// TwinCAT 3 PLC project Aufgabe5
// ProgramVersion: 3.1.4023.0
// libraries:
//   Tc2_Standard, * (Beckhoff Automation GmbH)
//   Tc2_System, * (Beckhoff Automation GmbH)
//   Tc3_Module, * (Beckhoff Automation GmbH)
// project tree:
//   / PlcTask.TcTTO
//   POUs/ Fb_EdgeDetector.TcPOU, FB_Integrator.TcPOU, FB_LowpassFilter.TcPOU, Fb_MeanCalculatorWForgettingFactor.TcPOU, FB_PWM.TcPOU (not stored), FB_SecondOrderHold.TcPOU, F_Sine.TcPOU, F_Square.TcPOU, MAIN.TcPOU
// real-time tasks:
//   TASK PlcTask: cycle T#10ms, priority 20, ADS port 350

CONFIGURATION Aufgabe5
    RESOURCE PLC ON TwinCAT3
        TASK PlcTask(INTERVAL := T#10ms, PRIORITY := 20);
        PROGRAM MAIN WITH PlcTask : MAIN;
    END_RESOURCE
END_CONFIGURATION

// ---- POUs/MAIN.TcPOU
PROGRAM MAIN
VAR
	// sinus
	u_k_sin			: REAL;				// u_k sinus
	u_k_sin_f		: REAL;				// u_k sinus filtered
	w_sin			: REAL := (1/tau);	// Frequenz
	lowPassSin		: FB_LowpassFilter;
	// constant
	u_k_cst			: REAL;				// u_k constant
	u_k_cst_f		: REAL;				// u_k constant filtered
	lowPassConst	: FB_LowpassFilter;
	// pt2
	d				: REAL		:= 0.2;
	w0				: REAL		:= 10;
	u_k_pt2_f		: REAL;				// u_k pt2 filtered
	secondOrder		: FB_SecondOrderHold;
	// integrator
	pwm				: FB_PWM;
	integrator		: FB_Integrator;
	dutyCyclePct	: REAL		:= 25; 	// duty cycle for PWM in %
	pwmOut			: REAL;				// pwm signal
	integratorOut	: REAL;				// integrated PWM signal
	
	actTime			: REAL 	:= 0;		// time increment
	
END_VAR
VAR CONSTANT
	sampleTime		: REAL	:= 0.001;	// Abtastzeit	
	tau 			: REAL	:= 0.1;		// filter constant
END_VAR

// Integrator PWM
pwm(dutyPct := dutyCyclePct, ymin := 0, ymax := 5, w := 3.14, t := actTime);
pwmOut := pwm.y;
integrator(u_k := pwmOut, T := sampleTime);
integratorOut := integrator.y_k;

// Lowpass Sinus
u_k_sin := F_Sine(A := 1.0, yoff := 0.0, w := w_sin, t := actTime);
lowPassSin(u_k := u_k_sin, T := sampleTime, tau := tau);
u_k_sin_f := lowPassSin.y_k;

// PT2 with sinus
secondOrder(u_k := u_k_sin, T := sampleTime, d := d, w0 := w0);
u_k_pt2_f := secondOrder.y_k;

actTime := actTime + sampleTime;

END_PROGRAM

// ---- POUs/FB_LowpassFilter.TcPOU
FUNCTION_BLOCK FB_LowpassFilter
VAR_INPUT
	u_k		: REAL;
	T		: REAL;
	tau		: REAL;
END_VAR
VAR_OUTPUT
	y_k		: REAL;
END_VAR
VAR
	y_k_1	: REAL;
END_VAR

// limit tau
IF tau < 0.0001 THEN
	tau := 0.0001;
END_IF

y_k := tau / (T+tau) * y_k_1 + T / (T+tau) * u_k;
y_k_1 := y_k;

END_FUNCTION_BLOCK

// ---- POUs/FB_SecondOrderHold.TcPOU
FUNCTION_BLOCK FB_SecondOrderHold
VAR_INPUT
	u_k		: REAL; // Eingangswert
	T		: REAL;	// Zeitkonstante
	d		: REAL; // Daempfung
	w0		: REAL; // Eigenfrequenz 
END_VAR
VAR_OUTPUT
	y_k		: REAL; // Ausgangswert
END_VAR
VAR
	a		: REAL; // Variable fuer w0^2 * T^2
	b 		: REAL; // Variable fuer 2 * d * w0 * T
	y_k_1	: REAL; // letzer Ausgangswert
	y_k_2	: REAL; // vorletzer Ausgangswert
END_VAR

a := (w0 * w0) * (T * T);
b := 2 * d * w0 * T; 

y_k := (u_k*a + 2*y_k_1 + b*y_k_1 - y_k_2) / (1 + b + a); 

y_k_2 := y_k_1;
y_k_1 := y_k;

END_FUNCTION_BLOCK

// ---- POUs/FB_Integrator.TcPOU
FUNCTION_BLOCK FB_Integrator
VAR_INPUT
	u_k		: REAL;
	T		: REAL;
END_VAR
VAR_OUTPUT
	y_k		: REAL;
END_VAR
VAR
	y_k_1	: REAL;
END_VAR

y_k := u_k * T + y_k_1;
y_k_1 := y_k;

END_FUNCTION_BLOCK

// ---- POUs/F_Sine.TcPOU
FUNCTION F_Sine : REAL
VAR_INPUT
	A		: REAL;	// Amplitude
	yoff	: REAL; // offset
	w		: REAL; // Kreisfrequenz (rad/s)
	t		: REAL; // Time (s)
END_VAR
VAR
END_VAR

F_Sine := (A * SIN(w*t)) + yoff;

END_FUNCTION

// ---- POUs/Fb_EdgeDetector.TcPOU
FUNCTION_BLOCK INTERNAL Fb_EdgeDetector
VAR_INPUT
	inputValue		: BOOL;
END_VAR
VAR_OUTPUT
	risingEdge		: BOOL;
	fallingEdge		: BOOL;
	doublePress		: BOOL;
	triplePress		: BOOL;
END_VAR
VAR
	i_risingEdgCnt			: INT := 0;  		// internal var
	lastValue 				: BOOL;				// last value registered
	tlastPush				: TIME := TIME();	// time when last push happened
	tLastRising				: TIME := TIME();	// time when last rising edge happened
	tDebounce	    		: TIME := T#20MS;   // time to debounce input value
	tMultiPressTime			: TIME := T#200MS;	// time between which multiple presses to allow the user to press button again
	
END_VAR

// reset output signals
fallingEdge := FALSE;
risingEdge := FALSE;
doublePress := FALSE;
triplePress := FALSE;

// if a change happened and new values get accepted
IF(inputValue <> lastValue AND (tlastPush + tDebounce) < TIME()) THEN
	IF(inputValue) THEN
		i_risingEdgCnt := i_risingEdgCnt + 1;
		
		tLastRising := TIME(); // reset last rising time (give another tMultiPressTime time to press the button another time
	ELSE
		fallingEdge := TRUE;
	END_IF
	lastValue := inputValue;  // overwrite stored value
	tlastPush := TIME();
END_IF


// handle rising edge (with double press)
CASE i_risingEdgCnt OF
	1:
	IF (tLastRising + tMultiPressTime) < TIME() THEN
		risingEdge := TRUE;
		i_risingEdgCnt := 0;
	END_IF
	
	2:
	IF (tLastRising + tMultiPressTime) < TIME() THEN
		doublePress := TRUE;
		i_risingEdgCnt := 0;
	END_IF
	
	3:
	// instantly report triple press, since no more amount of multi press is output
	triplePress := TRUE;
	i_risingEdgCnt := 0;
ELSE
	;
END_CASE

END_FUNCTION_BLOCK

// ---- POUs/Fb_MeanCalculatorWForgettingFactor.TcPOU
FUNCTION_BLOCK Fb_MeanCalculatorWForgettingFactor
VAR_IN_OUT
	r_inputValue			: REAL;
	r_forgettingFactor		: REAL;
END_VAR
VAR_OUTPUT
	r_meanValueOutput		: REAL;
END_VAR
VAR
	r_meanValue				: REAL;
	lr_numerator			: LREAL;
	lr_denominator			: LREAL;
	lr_forgFactorExp		: LREAL;
	i_counter				: DINT;
END_VAR

r_meanValue := (r_forgettingFactor * r_meanValue) + (1-r_forgettingFactor) * r_inputValue;
r_meanValueOutput := r_meanValue;

END_FUNCTION_BLOCK

// ---- POUs/F_Square.TcPOU
FUNCTION F_Square : REAL
VAR_INPUT
	ymin	: REAL;	// Minimalwert
	ymax	: REAL;	// Maximalwert
	yoff	: REAL; // offset
	w		: REAL; // Kreisfrequenz (rad/s)
	t		: REAL; // Time (s)
END_VAR
VAR
	sinRes	: REAL; // sine result
	squareRes: REAL;
END_VAR

sinRes := SIN(w*t);

IF (sinRes > 0) THEN
	squareRes := ymin;
ELSE
	squareRes := ymax;
END_IF

F_Square := squareRes + yoff;

END_FUNCTION
